FUNCTION F_Scaling : REAL
VAR_INPUT
	rawInput : INT;
END_VAR
VAR
END_VAR

F_Scaling := rawInput/327.67;

END_FUNCTION

(* stored: Version 1.1.0.1, ProductVersion 3.1.4024.12
   POU F_Scaling: Id {45ef72a9-5505-4f12-a785-64215dafa89f}, SpecialFunc None *)
